FUNCTION_BLOCK POU
VAR_INPUT
END_VAR
VAR_OUTPUT
END_VAR
VAR
END_VAR

END_FUNCTION_BLOCK

(* stored: Version 1.1.0.1, ProductVersion 3.1.4024.11
   POU POU: Id {b0522563-76c0-4877-999f-5efd3809bda5}, SpecialFunc None *)
